TYPE ST_CylinderX_Status :
    STRUCT
        Extended   : BOOL;
        Retracted  : BOOL;
        Extending  : BOOL;
        Retracting : BOOL;
    END_STRUCT
END_TYPE

(* stored: Version 1.1.0.1
   DUT ST_CylinderX_Status: Id {921932a2-6ed4-41dc-abc2-16e62097ddd3} *)
